PROGRAM AXIS_1
VAR
//Outputs: Power for Limit switches, Home Sensors, etc.
    //bPowerSwitchesAxis1 AT %Q*: BOOL:= TRUE;

//Hardware interlocks
    //bInterlockFwdOK AT %I*: BOOL;
END_VAR

//Initial parameters of an Axis
(*IF _TaskInfo[fbGetCurTaskIndex.index].FirstCycle THEN
    //Axis description for EPICS PV
    GVL.astAxes[1].stDescription.sAxisName := 'MotorApplication1';
    GVL.astAxes[1].stDescription.eUnit := E_AxisEngUnit.eMeter;
    GVL.astAxes[1].stDescription.nPrefix := -3;

    //Initial default values:
    GVL.astAxes[1].stConfig.eHomeSeq := 0;
    GVL.astAxes[1].stConfig.fHomePosition := 0.0;
    GVL.astAxes[1].stConfig.fHomeFinishDistance := 0.0;
    GVL.astAxes[1].stConfig.eRestorePosition := E_RestorePosition.eRestoreWithoutHome;
END_IF*)

//Define ACTIONS() or write exclusive code for an specific axis.
(*Eg. Stop when temperature reaches certain values, reduce speed if  a signal is activated, etc.
Eg. GVL.astAxes[x].stControl.bInterlockFwd := NOT bInterlockFwdOK;*)

//Limits for positive axis, Axis 1
IF astAxes[1].stStatus.fActPosition > 100 THEN
    SlitProg.mySlit.bPositiveAxis_FwdLimit := FALSE;
ELSE
     SlitProg.mySlit.bPositiveAxis_FwdLimit :=TRUE;
END_IF
IF astAxes[1].stStatus.fActPosition < -100 THEN
     SlitProg.mySlit.bPositiveAxis_BwdLimit :=FALSE;
ELSE
     SlitProg.mySlit.bPositiveAxis_BwdLimit :=TRUE;
END_IF

END_PROGRAM

(* stored: Version 1.1.0.1, ProductVersion 3.1.4024.11
   POU AXIS_1: Id {1e59798f-4551-4034-b486-d187e82e019a}, SpecialFunc None *)
